FUNCTION_BLOCK FB_TCIn
VAR_INPUT
	iMaxInCH : INT;
END_VAR
VAR_OUTPUT
END_VAR
VAR
	iIndex 		: INT;
	iMax		: INT;
END_VAR

IF iMaxInCH > GVL_Thermocouples.iTCchannelCount THEN
	iMax := GVL_Thermocouples.iTCchannelCount;
ELSE
	iMax := iMaxInCH;
END_IF

FOR iIndex :=1 TO iMax BY 1 DO 

	GVL_Thermocouples.hmi_config[iIndex].rTempC	:= TO_REAL(GVL_Thermocouples.hmi_config[iIndex].iRawCountIn)/10;
	GVL_Thermocouples.hmi_config[iIndex].rTempF	:=c_to_f
		(
		tempC:=GVL_Thermocouples.hmi_config[iIndex].rTempC
		);
END_FOR

END_FUNCTION_BLOCK

(* stored: Version 1.1.0.1, ProductVersion 3.1.4024.12
   POU FB_TCIn: Id {37959487-f699-46f5-9791-275b1b595234}, SpecialFunc None *)
